# EPICS substitutions: db/Beckhoff_5XXX/ecmcEL5131.substitutions
file "ecmcEL5131-chX.template"
{
    pattern {CH_ID}
            {01   }

}
